// TIA Portal V17 export
// export: Created 2024-08-07T21:44:03.571526Z, ExportSetting WithDefaults, DisplayName Totally Integrated Automation Portal, DisplayVersion V17 Update 7, DisplayName TIA Portal Openness, DisplayVersion V17 Update 7, DisplayName TIA Portal Version Control Interface, DisplayVersion V17, DisplayName SINAMICS Startdrive Advanced, DisplayVersion V17 SP2, DisplayName SINAMICS Startdrive G110M, G120, G120C, G120D, G120P, G115D, DisplayVersion V17 SP2, DisplayName SINAMICS Startdrive G130, G150, S120, S150, SINAMICS MV, S210, DisplayVersion V17 SP2, DisplayName STEP 7 Professional, DisplayVersion V17 Update 7, DisplayName STEP 7 Safety, DisplayVersion V17 Update 6, DisplayName WinCC Advanced / Unified PC, DisplayVersion V17 Update 7
DATA_BLOCK "DB_ProductionCountersList"   // DB65
{ S7_Optimized_Access := 'TRUE' }
VERSION : 0.1
// stored: AutoNumber true, DBAccessibleFromOPCUA true, DBAccessibleFromWebserver true, IsOnlyStoredInLoadMemory false, IsRetainMemResEnabled false, IsWriteProtectedInAS false, MemoryReserve 100
   VAR RETAIN
      Program { S7_SetPoint := 'True'} : Array[1.."NumberOfProductionPrograms"] of "UDT_ProductionProgramCounters";
      Machine : "UDT_Counters";
   END_VAR
BEGIN
   Program[1].Product[1].Shift[1..3].Ok := 0;
   Program[1].Product[2].Shift[1..3].Ok := 0;
   Program[1].Product[3].Shift[1..3].Ok := 0;
   Program[1].Product[4].Shift[1..3].Ok := 0;
   Program[1].Product[5].Shift[1..3].Ok := 0;
   Program[1].Product[6].Shift[1..3].Ok := 0;
   Program[1].Product[7].Shift[1..3].Ok := 0;
   Program[1].Product[8].Shift[1..3].Ok := 0;
   Program[2].Product[1].Shift[1..3].Ok := 0;
   Program[2].Product[2].Shift[1..3].Ok := 0;
   Program[2].Product[3].Shift[1..3].Ok := 0;
   Program[2].Product[4].Shift[1..3].Ok := 0;
   Program[2].Product[5].Shift[1..3].Ok := 0;
   Program[2].Product[6].Shift[1..3].Ok := 0;
   Program[2].Product[7].Shift[1..3].Ok := 0;
   Program[2].Product[8].Shift[1..3].Ok := 0;
   Program[3].Product[1].Shift[1..3].Ok := 0;
   Program[3].Product[2].Shift[1..3].Ok := 0;
   Program[3].Product[3].Shift[1..3].Ok := 0;
   Program[3].Product[4].Shift[1..3].Ok := 0;
   Program[3].Product[5].Shift[1..3].Ok := 0;
   Program[3].Product[6].Shift[1..3].Ok := 0;
   Program[3].Product[7].Shift[1..3].Ok := 0;
   Program[3].Product[8].Shift[1..3].Ok := 0;
   Program[4].Product[1].Shift[1..3].Ok := 0;
   Program[4].Product[2].Shift[1..3].Ok := 0;
   Program[4].Product[3].Shift[1..3].Ok := 0;
   Program[4].Product[4].Shift[1..3].Ok := 0;
   Program[4].Product[5].Shift[1..3].Ok := 0;
   Program[4].Product[6].Shift[1..3].Ok := 0;
   Program[4].Product[7].Shift[1..3].Ok := 0;
   Program[4].Product[8].Shift[1..3].Ok := 0;
   Program[5].Product[1].Shift[1..3].Ok := 0;
   Program[5].Product[2].Shift[1..3].Ok := 0;
   Program[5].Product[3].Shift[1..3].Ok := 0;
   Program[5].Product[4].Shift[1..3].Ok := 0;
   Program[5].Product[5].Shift[1..3].Ok := 0;
   Program[5].Product[6].Shift[1..3].Ok := 0;
   Program[5].Product[7].Shift[1..3].Ok := 0;
   Program[5].Product[8].Shift[1..3].Ok := 0;
   Program[6].Product[1].Shift[1..3].Ok := 0;
   Program[6].Product[2].Shift[1..3].Ok := 0;
   Program[6].Product[3].Shift[1..3].Ok := 0;
   Program[6].Product[4].Shift[1..3].Ok := 0;
   Program[6].Product[5].Shift[1..3].Ok := 0;
   Program[6].Product[6].Shift[1..3].Ok := 0;
   Program[6].Product[7].Shift[1..3].Ok := 0;
   Program[6].Product[8].Shift[1..3].Ok := 0;
   Program[7].Product[1].Shift[1..3].Ok := 0;
   Program[7].Product[2].Shift[1..3].Ok := 0;
   Program[7].Product[3].Shift[1..3].Ok := 0;
   Program[7].Product[4].Shift[1..3].Ok := 0;
   Program[7].Product[5].Shift[1..3].Ok := 0;
   Program[7].Product[6].Shift[1..3].Ok := 0;
   Program[7].Product[7].Shift[1..3].Ok := 0;
   Program[7].Product[8].Shift[1..3].Ok := 0;
   Program[8].Product[1].Shift[1..3].Ok := 0;
   Program[8].Product[2].Shift[1..3].Ok := 0;
   Program[8].Product[3].Shift[1..3].Ok := 0;
   Program[8].Product[4].Shift[1..3].Ok := 0;
   Program[8].Product[5].Shift[1..3].Ok := 0;
   Program[8].Product[6].Shift[1..3].Ok := 0;
   Program[8].Product[7].Shift[1..3].Ok := 0;
   Program[8].Product[8].Shift[1..3].Ok := 0;
   Program[1].Product[1].Shift[1..3].Nok := 0;
   Program[1].Product[2].Shift[1..3].Nok := 0;
   Program[1].Product[3].Shift[1..3].Nok := 0;
   Program[1].Product[4].Shift[1..3].Nok := 0;
   Program[1].Product[5].Shift[1..3].Nok := 0;
   Program[1].Product[6].Shift[1..3].Nok := 0;
   Program[1].Product[7].Shift[1..3].Nok := 0;
   Program[1].Product[8].Shift[1..3].Nok := 0;
   Program[2].Product[1].Shift[1..3].Nok := 0;
   Program[2].Product[2].Shift[1..3].Nok := 0;
   Program[2].Product[3].Shift[1..3].Nok := 0;
   Program[2].Product[4].Shift[1..3].Nok := 0;
   Program[2].Product[5].Shift[1..3].Nok := 0;
   Program[2].Product[6].Shift[1..3].Nok := 0;
   Program[2].Product[7].Shift[1..3].Nok := 0;
   Program[2].Product[8].Shift[1..3].Nok := 0;
   Program[3].Product[1].Shift[1..3].Nok := 0;
   Program[3].Product[2].Shift[1..3].Nok := 0;
   Program[3].Product[3].Shift[1..3].Nok := 0;
   Program[3].Product[4].Shift[1..3].Nok := 0;
   Program[3].Product[5].Shift[1..3].Nok := 0;
   Program[3].Product[6].Shift[1..3].Nok := 0;
   Program[3].Product[7].Shift[1..3].Nok := 0;
   Program[3].Product[8].Shift[1..3].Nok := 0;
   Program[4].Product[1].Shift[1..3].Nok := 0;
   Program[4].Product[2].Shift[1..3].Nok := 0;
   Program[4].Product[3].Shift[1..3].Nok := 0;
   Program[4].Product[4].Shift[1..3].Nok := 0;
   Program[4].Product[5].Shift[1..3].Nok := 0;
   Program[4].Product[6].Shift[1..3].Nok := 0;
   Program[4].Product[7].Shift[1..3].Nok := 0;
   Program[4].Product[8].Shift[1..3].Nok := 0;
   Program[5].Product[1].Shift[1..3].Nok := 0;
   Program[5].Product[2].Shift[1..3].Nok := 0;
   Program[5].Product[3].Shift[1..3].Nok := 0;
   Program[5].Product[4].Shift[1..3].Nok := 0;
   Program[5].Product[5].Shift[1..3].Nok := 0;
   Program[5].Product[6].Shift[1..3].Nok := 0;
   Program[5].Product[7].Shift[1..3].Nok := 0;
   Program[5].Product[8].Shift[1..3].Nok := 0;
   Program[6].Product[1].Shift[1..3].Nok := 0;
   Program[6].Product[2].Shift[1..3].Nok := 0;
   Program[6].Product[3].Shift[1..3].Nok := 0;
   Program[6].Product[4].Shift[1..3].Nok := 0;
   Program[6].Product[5].Shift[1..3].Nok := 0;
   Program[6].Product[6].Shift[1..3].Nok := 0;
   Program[6].Product[7].Shift[1..3].Nok := 0;
   Program[6].Product[8].Shift[1..3].Nok := 0;
   Program[7].Product[1].Shift[1..3].Nok := 0;
   Program[7].Product[2].Shift[1..3].Nok := 0;
   Program[7].Product[3].Shift[1..3].Nok := 0;
   Program[7].Product[4].Shift[1..3].Nok := 0;
   Program[7].Product[5].Shift[1..3].Nok := 0;
   Program[7].Product[6].Shift[1..3].Nok := 0;
   Program[7].Product[7].Shift[1..3].Nok := 0;
   Program[7].Product[8].Shift[1..3].Nok := 0;
   Program[8].Product[1].Shift[1..3].Nok := 0;
   Program[8].Product[2].Shift[1..3].Nok := 0;
   Program[8].Product[3].Shift[1..3].Nok := 0;
   Program[8].Product[4].Shift[1..3].Nok := 0;
   Program[8].Product[5].Shift[1..3].Nok := 0;
   Program[8].Product[6].Shift[1..3].Nok := 0;
   Program[8].Product[7].Shift[1..3].Nok := 0;
   Program[8].Product[8].Shift[1..3].Nok := 0;
   Program[1].Product[1].Overall.Ok := 62;
   Program[1].Product[2..8].Overall.Ok := 0;
   Program[2].Product[1].Overall.Ok := 32;
   Program[2].Product[2..8].Overall.Ok := 0;
   Program[3].Product[1..8].Overall.Ok := 0;
   Program[4].Product[1..8].Overall.Ok := 0;
   Program[5].Product[1].Overall.Ok := 141;
   Program[5].Product[2..8].Overall.Ok := 0;
   Program[6].Product[1].Overall.Ok := 40;
   Program[6].Product[2..8].Overall.Ok := 0;
   Program[7].Product[1].Overall.Ok := 50;
   Program[7].Product[2..8].Overall.Ok := 0;
   Program[8].Product[1..8].Overall.Ok := 0;
   Program[1].Product[1].Overall.Nok := 9;
   Program[1].Product[2..8].Overall.Nok := 0;
   Program[2].Product[1].Overall.Nok := 7;
   Program[2].Product[2..8].Overall.Nok := 0;
   Program[3].Product[1..8].Overall.Nok := 0;
   Program[4].Product[1..8].Overall.Nok := 0;
   Program[5].Product[1].Overall.Nok := 43;
   Program[5].Product[2..8].Overall.Nok := 0;
   Program[6].Product[1].Overall.Nok := 3;
   Program[6].Product[2..8].Overall.Nok := 0;
   Program[7].Product[1..8].Overall.Nok := 0;
   Program[8].Product[1..8].Overall.Nok := 0;
   Machine.Ok := 325;
   Machine.Nok := 62;
END_DATA_BLOCK
